# EPICS substitutions: ssaApp/Db/gunCommon.substitutions
# Common controls for gun SSAs.
# Macros:
#   OUT: PV attribute
#   MASK: Bitmask to select which SSAs to control; e.g. 3 for SSAs 1 & 2, 15 for SSAs 1,2,3,4.
#   DLY: Delay between sequence steps

file "ssaCommonControls_2x.template" {
pattern
{SSA1  SSA2,  N,  M,        OUT,  DLY}
{SSA1, SSA2, "", "",    PowerOn,  1.0}
{SSA1, SSA2, "", "",   PowerOff,  0.1}
{SSA1, SSA2, "", "", FaultReset,  1.0}
}
